// TIA Portal V18 export
// export: Created 2025-12-01T12:38:08.5332693Z, ExportSetting None, DisplayName Totally Integrated Automation Portal, DisplayVersion V18 Update 5, DisplayName TIA Portal Openness, DisplayVersion V18 Update 5, DisplayName TIA Portal Teamcenter Gateway, DisplayVersion V18, DisplayName TIA Portal Version Control Interface, DisplayVersion V18, DisplayName STEP 7 Professional, DisplayVersion V18 Update 5, DisplayName STEP 7 Safety, DisplayVersion V18, DisplayName WinCC Professional, DisplayVersion V18 Update 5
DATA_BLOCK "ST10_Flow23_KReserveLifting_iDB"   // DB1093
// stored: AutoNumber false, InstanceOfName ST10_Flow23_KReserveLifting, InstanceOfType FB
"ST10_Flow23_KReserveLifting"
   // // inherited from GRAPH_BASE
   // VAR_INPUT
   //    iSysInface : "RCS_SysComInterface_V1";
   // END_VAR
   // VAR_IN_OUT
   //    ioPM_Inface : "RCS_PMInterface_V1";
   //    ioStatus : Int;
   // END_VAR
   // VAR
   //    sCtrlMode { S7_SetPoint := 'True'} : "SysFlowCtrlGraph";
   //    sUpdMES_Data : Bool;
   //    工件放行中 : Bool;
   //    前站站号 { ExternalAccessible := 'False'; ExternalVisible := 'False'; ExternalWritable := 'False'} : UInt;
   //    本站站号 { ExternalAccessible := 'False'; ExternalVisible := 'False'; ExternalWritable := 'False'} : UInt;
   //    弹窗Temp : Array[1..10] of Int;
   //    AlarmID : Int;
   //    TON { S7_SetPoint := 'True'} : Array[0..10] of TON_TIME;
   //    TOF { S7_SetPoint := 'True'} : Array[0..10] of TOF_TIME;
   //    sUP { S7_SetPoint := 'True'} : Array[0..10] of Bool;
   //    更新RFID完成 : Bool;
   //    RT_DATA { ExternalAccessible := 'False'; ExternalVisible := 'False'; ExternalWritable := 'False'; S7_SetPoint := 'True'} : G7_RTDataPlus_V6;
   //    Trans1 { ExternalAccessible := 'False'; ExternalVisible := 'False'; ExternalWritable := 'False'; S7_SetPoint := 'True'} : G7_TransitionPlus_V6;
   //    Trans2 { ExternalAccessible := 'False'; ExternalVisible := 'False'; ExternalWritable := 'False'; S7_SetPoint := 'True'} : G7_TransitionPlus_V6;
   //    Trans3 { ExternalAccessible := 'False'; ExternalVisible := 'False'; ExternalWritable := 'False'; S7_SetPoint := 'True'} : G7_TransitionPlus_V6;
   //    Trans325 { ExternalAccessible := 'False'; ExternalVisible := 'False'; ExternalWritable := 'False'; S7_SetPoint := 'True'} : G7_TransitionPlus_V6;
   //    Trans10 { ExternalAccessible := 'False'; ExternalVisible := 'False'; ExternalWritable := 'False'; S7_SetPoint := 'True'} : G7_TransitionPlus_V6;
   //    Trans102 { ExternalAccessible := 'False'; ExternalVisible := 'False'; ExternalWritable := 'False'; S7_SetPoint := 'True'} : G7_TransitionPlus_V6;
   //    Trans22 { ExternalAccessible := 'False'; ExternalVisible := 'False'; ExternalWritable := 'False'; S7_SetPoint := 'True'} : G7_TransitionPlus_V6;
   //    Trans23 { ExternalAccessible := 'False'; ExternalVisible := 'False'; ExternalWritable := 'False'; S7_SetPoint := 'True'} : G7_TransitionPlus_V6;
   //    Trans24 { ExternalAccessible := 'False'; ExternalVisible := 'False'; ExternalWritable := 'False'; S7_SetPoint := 'True'} : G7_TransitionPlus_V6;
   //    Trans25 { ExternalAccessible := 'False'; ExternalVisible := 'False'; ExternalWritable := 'False'; S7_SetPoint := 'True'} : G7_TransitionPlus_V6;
   //    Trans27 { ExternalAccessible := 'False'; ExternalVisible := 'False'; ExternalWritable := 'False'; S7_SetPoint := 'True'} : G7_TransitionPlus_V6;
   //    Trans28 { ExternalAccessible := 'False'; ExternalVisible := 'False'; ExternalWritable := 'False'; S7_SetPoint := 'True'} : G7_TransitionPlus_V6;
   //    Trans29 { ExternalAccessible := 'False'; ExternalVisible := 'False'; ExternalWritable := 'False'; S7_SetPoint := 'True'} : G7_TransitionPlus_V6;
   //    Trans30 { ExternalAccessible := 'False'; ExternalVisible := 'False'; ExternalWritable := 'False'; S7_SetPoint := 'True'} : G7_TransitionPlus_V6;
   //    Trans31 { ExternalAccessible := 'False'; ExternalVisible := 'False'; ExternalWritable := 'False'; S7_SetPoint := 'True'} : G7_TransitionPlus_V6;
   //    Trans32 { ExternalAccessible := 'False'; ExternalVisible := 'False'; ExternalWritable := 'False'; S7_SetPoint := 'True'} : G7_TransitionPlus_V6;
   //    Trans33 { ExternalAccessible := 'False'; ExternalVisible := 'False'; ExternalWritable := 'False'; S7_SetPoint := 'True'} : G7_TransitionPlus_V6;
   //    Trans34 { ExternalAccessible := 'False'; ExternalVisible := 'False'; ExternalWritable := 'False'; S7_SetPoint := 'True'} : G7_TransitionPlus_V6;
   //    Trans35 { ExternalAccessible := 'False'; ExternalVisible := 'False'; ExternalWritable := 'False'; S7_SetPoint := 'True'} : G7_TransitionPlus_V6;
   //    Trans36 { ExternalAccessible := 'False'; ExternalVisible := 'False'; ExternalWritable := 'False'; S7_SetPoint := 'True'} : G7_TransitionPlus_V6;
   //    Trans200 { ExternalAccessible := 'False'; ExternalVisible := 'False'; ExternalWritable := 'False'; S7_SetPoint := 'True'} : G7_TransitionPlus_V6;
   //    Trans765 { ExternalAccessible := 'False'; ExternalVisible := 'False'; ExternalWritable := 'False'; S7_SetPoint := 'True'} : G7_TransitionPlus_V6;
   //    Trans117 { ExternalAccessible := 'False'; ExternalVisible := 'False'; ExternalWritable := 'False'; S7_SetPoint := 'True'} : G7_TransitionPlus_V6;
   //    Trans119 { ExternalAccessible := 'False'; ExternalVisible := 'False'; ExternalWritable := 'False'; S7_SetPoint := 'True'} : G7_TransitionPlus_V6;
   //    Trans772 { ExternalAccessible := 'False'; ExternalVisible := 'False'; ExternalWritable := 'False'; S7_SetPoint := 'True'} : G7_TransitionPlus_V6;
   //    Trans773 { ExternalAccessible := 'False'; ExternalVisible := 'False'; ExternalWritable := 'False'; S7_SetPoint := 'True'} : G7_TransitionPlus_V6;
   //    Trans136 { ExternalAccessible := 'False'; ExternalVisible := 'False'; ExternalWritable := 'False'; S7_SetPoint := 'True'} : G7_TransitionPlus_V6;
   //    Trans774 { ExternalAccessible := 'False'; ExternalVisible := 'False'; ExternalWritable := 'False'; S7_SetPoint := 'True'} : G7_TransitionPlus_V6;
   //    Trans775 { ExternalAccessible := 'False'; ExternalVisible := 'False'; ExternalWritable := 'False'; S7_SetPoint := 'True'} : G7_TransitionPlus_V6;
   //    Trans139 { ExternalAccessible := 'False'; ExternalVisible := 'False'; ExternalWritable := 'False'; S7_SetPoint := 'True'} : G7_TransitionPlus_V6;
   //    Trans140 { ExternalAccessible := 'False'; ExternalVisible := 'False'; ExternalWritable := 'False'; S7_SetPoint := 'True'} : G7_TransitionPlus_V6;
   //    Trans776 { ExternalAccessible := 'False'; ExternalVisible := 'False'; ExternalWritable := 'False'; S7_SetPoint := 'True'} : G7_TransitionPlus_V6;
   //    Trans142 { ExternalAccessible := 'False'; ExternalVisible := 'False'; ExternalWritable := 'False'; S7_SetPoint := 'True'} : G7_TransitionPlus_V6;
   //    Trans777 { ExternalAccessible := 'False'; ExternalVisible := 'False'; ExternalWritable := 'False'; S7_SetPoint := 'True'} : G7_TransitionPlus_V6;
   //    Trans141 { ExternalAccessible := 'False'; ExternalVisible := 'False'; ExternalWritable := 'False'; S7_SetPoint := 'True'} : G7_TransitionPlus_V6;
   //    Trans250 { ExternalAccessible := 'False'; ExternalVisible := 'False'; ExternalWritable := 'False'; S7_SetPoint := 'True'} : G7_TransitionPlus_V6;
   //    Trans613 { ExternalAccessible := 'False'; ExternalVisible := 'False'; ExternalWritable := 'False'; S7_SetPoint := 'True'} : G7_TransitionPlus_V6;
   //    F23_Initial { ExternalAccessible := 'False'; ExternalVisible := 'False'; ExternalWritable := 'False'; S7_SetPoint := 'True'} : G7_StepPlus_V6;
   //    S2 { ExternalAccessible := 'False'; ExternalVisible := 'False'; ExternalWritable := 'False'; S7_SetPoint := 'True'} : G7_StepPlus_V6;
   //    S3 { ExternalAccessible := 'False'; ExternalVisible := 'False'; ExternalWritable := 'False'; S7_SetPoint := 'True'} : G7_StepPlus_V6;
   //    S4 { ExternalAccessible := 'False'; ExternalVisible := 'False'; ExternalWritable := 'False'; S7_SetPoint := 'True'} : G7_StepPlus_V6;
   //    S5_MESInitial { ExternalAccessible := 'False'; ExternalVisible := 'False'; ExternalWritable := 'False'; S7_SetPoint := 'True'} : G7_StepPlus_V6;
   //    WaitRobotInitialFinish { ExternalAccessible := 'False'; ExternalVisible := 'False'; ExternalWritable := 'False'; S7_SetPoint := 'True'} : G7_StepPlus_V6;
   //    S10_InitialFinish { ExternalAccessible := 'False'; ExternalVisible := 'False'; ExternalWritable := 'False'; S7_SetPoint := 'True'} : G7_StepPlus_V6;
   //    StatusError { ExternalAccessible := 'False'; ExternalVisible := 'False'; ExternalWritable := 'False'; S7_SetPoint := 'True'} : G7_StepPlus_V6;
   //    CheckStopPalletExist { ExternalAccessible := 'False'; ExternalVisible := 'False'; ExternalWritable := 'False'; S7_SetPoint := 'True'} : G7_StepPlus_V6;
   //    TimeDelay { ExternalAccessible := 'False'; ExternalVisible := 'False'; ExternalWritable := 'False'; S7_SetPoint := 'True'} : G7_StepPlus_V6;
   //    MotorCCWStart { ExternalAccessible := 'False'; ExternalVisible := 'False'; ExternalWritable := 'False'; S7_SetPoint := 'True'} : G7_StepPlus_V6;
   //    MotorCWStart { ExternalAccessible := 'False'; ExternalVisible := 'False'; ExternalWritable := 'False'; S7_SetPoint := 'True'} : G7_StepPlus_V6;
   //    ProcessStart { ExternalAccessible := 'False'; ExternalVisible := 'False'; ExternalWritable := 'False'; S7_SetPoint := 'True'} : G7_StepPlus_V6;
   //    "H-shaftLiftingLiftingCylinderToWP" { ExternalAccessible := 'False'; ExternalVisible := 'False'; ExternalWritable := 'False'; S7_SetPoint := 'True'} : G7_StepPlus_V6;
   //    CheckShaftLiftingCylinderPos { ExternalAccessible := 'False'; ExternalVisible := 'False'; ExternalWritable := 'False'; S7_SetPoint := 'True'} : G7_StepPlus_V6;
   //    "K-reserveLifting3PalletLocationCylindertoHP" { ExternalAccessible := 'False'; ExternalVisible := 'False'; ExternalWritable := 'False'; S7_SetPoint := 'True'} : G7_StepPlus_V6;
   //    "K-reserveLifting3PalletLocationCylindertoWP_1" { ExternalAccessible := 'False'; ExternalVisible := 'False'; ExternalWritable := 'False'; S7_SetPoint := 'True'} : G7_StepPlus_V6;
   //    Step131 { ExternalAccessible := 'False'; ExternalVisible := 'False'; ExternalWritable := 'False'; S7_SetPoint := 'True'} : G7_StepPlus_V6;
   //    MotorStop { ExternalAccessible := 'False'; ExternalVisible := 'False'; ExternalWritable := 'False'; S7_SetPoint := 'True'} : G7_StepPlus_V6;
   //    CheckPalletExist { ExternalAccessible := 'False'; ExternalVisible := 'False'; ExternalWritable := 'False'; S7_SetPoint := 'True'} : G7_StepPlus_V6;
   //    RequestRobotPickPallet { ExternalAccessible := 'False'; ExternalVisible := 'False'; ExternalWritable := 'False'; S7_SetPoint := 'True'} : G7_StepPlus_V6;
   //    WaitingPalletUnloading { ExternalAccessible := 'False'; ExternalVisible := 'False'; ExternalWritable := 'False'; S7_SetPoint := 'True'} : G7_StepPlus_V6;
   //    PalletRequest { ExternalAccessible := 'False'; ExternalVisible := 'False'; ExternalWritable := 'False'; S7_SetPoint := 'True'} : G7_StepPlus_V6;
   //    RobotCountClear0 { ExternalAccessible := 'False'; ExternalVisible := 'False'; ExternalWritable := 'False'; S7_SetPoint := 'True'} : G7_StepPlus_V6;
   //    "K-reserveLifting3PalletLocationCylindertoHP_2" { ExternalAccessible := 'False'; ExternalVisible := 'False'; ExternalWritable := 'False'; S7_SetPoint := 'True'} : G7_StepPlus_V6;
   //    "K-reserveLifting3PalletLocationCylindertoHP_3" { ExternalAccessible := 'False'; ExternalVisible := 'False'; ExternalWritable := 'False'; S7_SetPoint := 'True'} : G7_StepPlus_V6;
   //    MotorCCWRun { ExternalAccessible := 'False'; ExternalVisible := 'False'; ExternalWritable := 'False'; S7_SetPoint := 'True'} : G7_StepPlus_V6;
   //    "Motor Stop" { ExternalAccessible := 'False'; ExternalVisible := 'False'; ExternalWritable := 'False'; S7_SetPoint := 'True'} : G7_StepPlus_V6;
   //    "K-reserveLiftingCylindertoWP_4" { ExternalAccessible := 'False'; ExternalVisible := 'False'; ExternalWritable := 'False'; S7_SetPoint := 'True'} : G7_StepPlus_V6;
   //    "K-reserveLifting3PalletLocationCylindertoHP_4" { ExternalAccessible := 'False'; ExternalVisible := 'False'; ExternalWritable := 'False'; S7_SetPoint := 'True'} : G7_StepPlus_V6;
   //    MotorCCWRun_1 { ExternalAccessible := 'False'; ExternalVisible := 'False'; ExternalWritable := 'False'; S7_SetPoint := 'True'} : G7_StepPlus_V6;
   //    "Process Finish" { ExternalAccessible := 'False'; ExternalVisible := 'False'; ExternalWritable := 'False'; S7_SetPoint := 'True'} : G7_StepPlus_V6;
   // END_VAR
BEGIN
END_DATA_BLOCK
